TYPE (* IEC61131-3, Table 14#5 *)
  (* Standard: 1131-3 *)
  (* Version 0.0, 10/1/2026, Schneider Electric, Template *)
  PACKAGE Main;
  {SET_ATTRIBUTE(nxtDataType, RnsWMfuluD/126BLvQqwGkV6QmDNh3dwnLKmeFT5+q+cN9sWJNGV/yJwVCpVSucD1tGLYM4OnBXYgkCt7CDTMTMdcaPdDmWz9Gr9yqb1auO6DhN/811gPwZegzo+YN9HUJM+RBxfMAI=)}
  dtStruct : STRUCT
    A : INT;
    B : REAL;
    C : STRING[20];
    D : BOOL;
  END_STRUCT;
END_TYPE
